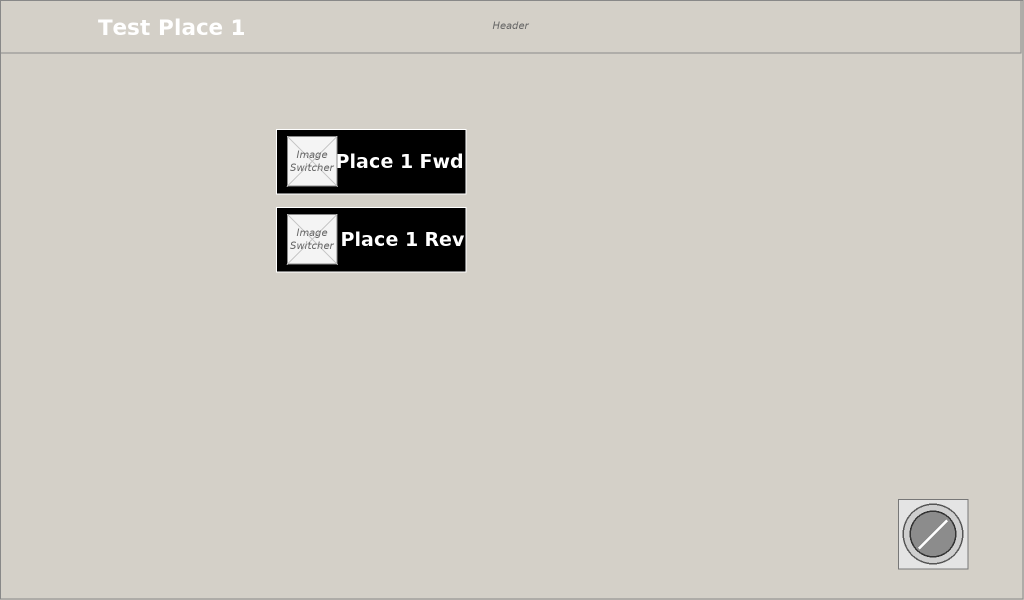
VISUALIZATION Test_Place1  // 1024x600
    Frame (0,-2 1021x55)
        shows Header()
    Label (95,15 250x25), "Test Place 1"
    RotarySwitch (898,499 70x70), variable: HMI_GVL.bTestModeEnablePlacing1, behaviour: TOGGLE, style: Switch-RotarySwitch-Gray
    RoundedRectangle (276,129 190x65)
        toggle Status_GVL.stMotor_Placing1.iTestForward
    Label (331,149 137x25), "Place 1 Fwd"
    ImageSwitcher (287,136 50x50), variable: Status_GVL.stMotor_Placing1.iTestForward, behaviour: TOGGLE
    RoundedRectangle (276,207 190x65)
        toggle Status_GVL.stMotor_Placing1.iTestReverse
    Label (334,227 137x25), "Place 1 Rev"
    ImageSwitcher (287,214 50x50), variable: Status_GVL.stMotor_Placing1.iTestReverse, behaviour: TOGGLE
END_VISUALIZATION

(* stored: Version 1.1.0.1, ProductVersion 3.1.4024.12
   Visu Test_Place1: Id {b2217a9c-bba3-498a-8c88-e78470e0aec4} *)
